(* IEC 61131-3 sources: VFDLib/, 12 files *)

(* ---- VFD.typ ---- *)
(********************************************************************
 * COPYRIGHT -- Automation Resources Group
 ********************************************************************
 * Library: VFDLib
 * File: VFD.typ
 * Author: David Blackburn
 * Created: December 21, 2011
 ********************************************************************
 * Data types of library VFDLib
 ********************************************************************)

TYPE
	VFD_ST_enum :
		(
		VFD_ST_NOTRDYTOSWON := 1,
		VFD_ST_SWONDISABLED,
		VFD_ST_RDYTOSWON,
		VFD_ST_SWON,
		VFD_ST_ENABLED,
		VFD_ST_QUICKSTOPACTIVE,
		VFD_ST_FAULTRXNACTIVE,
		VFD_ST_FAULT,
		VFD_ST_
		);
	VFD_Internal_typ : 	STRUCT
		ScaleIn : Scale_typ;
		ScaleOut : Scale_typ;
		AckResetTimer : TON;
		CMD : VFD_IN_CMD_typ;
	END_STRUCT;
	VFD_TEST_STAT_typ : 	STRUCT
		ActualVelocity : REAL;
		ActualVelocity_RPM : REAL;
		Error : BOOL;
		ErrorID : UINT;
		ErrorString : STRING[VFD_STRLEN_ERROR];
		RdyToSwOn : BOOL;
		SwOn : BOOL;
		OpEnabled : BOOL;
		Fault : BOOL;
		FaultID : UINT;
		VoltageDisabled : BOOL;
		QuickStop : BOOL;
		SwOnDisabled : BOOL;
		AlarmPresent : BOOL;
		RefReached : BOOL;
		State : DINT;
	END_STRUCT;
	VFD_TEST_typ : 	STRUCT
		Enable : BOOL;
		CMD : VFD_IN_CMD_typ;
		PAR : VFD_IN_PAR_typ;
		STAT : VFD_TEST_STAT_typ;
	END_STRUCT;
	VFD_OUT_STAT_Extended_typ : 	STRUCT
		Running : BOOL;
		DCInjection : BOOL;
		Transient : BOOL;
		ThermalOverloadAlarm : BOOL;
		BrakeAlarm : BOOL;
		Accelerating : BOOL;
		Decelerating : BOOL;
		CurrentLimitAlarm : BOOL;
		FastStop : BOOL;
		DirectionReq : BOOL;
	END_STRUCT;
	VFD_OUT_STAT_DriveStatus_typ : 	STRUCT
		RdyToSwOn : BOOL;
		SwOn : BOOL;
		OpEnabled : BOOL;
		Fault : BOOL;
		FaultID : UINT;
		FaultString : STRING[VFD_STRLEN_ERROR];
		VoltageDisabled : BOOL;
		QuickStop : BOOL;
		SwOnDisabled : BOOL;
		AlarmPresent : BOOL;
		RefReached : BOOL;
		RefExceeded : BOOL;
		StopKey : BOOL;
		DirectionOut : BOOL;
	END_STRUCT;
	VFD_OUT_STAT_typ : 	STRUCT
		ActualVelocity : REAL;
		ActualVelocity_RPM : REAL;
		DriveStatus : VFD_OUT_STAT_DriveStatus_typ;
		Extended : VFD_OUT_STAT_Extended_typ;
		State : DINT;
		Error : BOOL;
		ErrorID : UINT;
		ErrorString : STRING[VFD_STRLEN_ERROR];
	END_STRUCT;
	VFD_OUT_typ : 	STRUCT
		STAT : VFD_OUT_STAT_typ;
	END_STRUCT;
	VFD_IN_CFG_Scale_typ : 	STRUCT
		MinUnits : REAL;
		MinRPM : REAL;
		MaxUnits : REAL;
		MaxRPM : REAL;
	END_STRUCT;
	VFD_IN_CFG_typ : 	STRUCT
		Scale : VFD_IN_CFG_Scale_typ; (*2-point motor speed scaling*)
	END_STRUCT;
	VFD_IN_PAR_typ : 	STRUCT
		Velocity : REAL; (*Set motor speed in units.*)
	END_STRUCT;
	VFD_IN_CMD_typ : 	STRUCT
		Power : BOOL; (*Enable motor output*)
		Run : BOOL; (*Run motor at speed*)
		Reverse : BOOL; (*Run in reverse (must also set Run for motion)*)
		AcknowledgeError : BOOL; (*Reset drive faults*)
		Restart : BOOL; (*Restart drive after recovering from a fault*)
	END_STRUCT;
	VFD_IN_typ : 	STRUCT
		CMD : VFD_IN_CMD_typ;
		PAR : VFD_IN_PAR_typ;
		CFG : VFD_IN_CFG_typ;
	END_STRUCT;
	VFD_typ : 	STRUCT
		IN : VFD_IN_typ;
		OUT : VFD_OUT_typ;
		TEST : VFD_TEST_typ;
		IOMap : VFD_IO_typ;
		Encoder : VFD_Encoder_typ;
		Internal : VFD_Internal_typ;
	END_STRUCT;
END_TYPE

(* ---- VFD_IO.typ ---- *)
(*
 * File: VFD_IO.typ
 * Copyright (c) 2023 Loupe
 * https://loupe.team
 *
 * This file is part of VFDLib, licensed under the MIT License.
 *
 *)

TYPE
	VFD_IO_OUT_typ : 	STRUCT
		CMDD_Output : UINT;
		CMI_Output : UINT;
		LFRD_Output : INT;
		IOLR_Output_Bool : ARRAY[0..9] OF BOOL;
		DigitalOutput01 : BOOL;
		EnableCounter : BOOL;
	END_STRUCT;
	VFD_IO_IN_ModuleInfo_typ : 	STRUCT
		SerialNumber : UDINT;
		ModuleID : UINT;
		HardwareVariant : UINT;
		FirmwareVersion : UINT;
		ACPi_ModuleID : UDINT;
		ACPi_SerialNumber : UDINT;
	END_STRUCT;
	VFD_IO_IN_typ : 	STRUCT
		ModuleOK : BOOL;
		ModuleInfo : VFD_IO_IN_ModuleInfo_typ;
		ETAD_Input : UINT;
		ETI_Input : UINT;
		RFRD_Input : INT;
		OTR_Input : INT;
		LCR_Input : UINT;
		THD_Input : UINT;
		THR_Input : UINT;
		IOLR_Input_Bool : ARRAY[0..9] OF BOOL;
		ERRD_Input : UINT;
		LFT_Input : INT;
		StatusDigitalOutput01 : BOOL;
		Counter : DINT;
	END_STRUCT;
	VFD_IO_typ : 	STRUCT
		IN : VFD_IO_IN_typ;
		OUT : VFD_IO_OUT_typ;
	END_STRUCT;
END_TYPE

(* ---- VFDEncoder.typ ---- *)
(*
 * File: VFDEncoder.typ
 * Copyright (c) 2023 Loupe
 * https://loupe.team
 *
 * This file is part of VFDLib, licensed under the MIT License.
 *
 *)

TYPE
	VFD_Encoder_Internal_typ : 	STRUCT
		RTInfo : RTInfo;
		SpeedEst : SpeedEst;
		ScaleOut : Scale_typ;
	END_STRUCT;
	VFD_Encoder_OUT_STAT_typ : 	STRUCT
		Error : BOOL;
	END_STRUCT;
	VFD_Encoder_OUT_typ : 	STRUCT
		SpeedUnits : REAL;
		SpeedCounts : REAL;
		STAT : VFD_Encoder_OUT_STAT_typ;
	END_STRUCT;
	VFD_Encoder_IN_CFG_Scale_typ : 	STRUCT
		MinUnits : REAL;
		MinCounts : REAL;
		MaxUnits : REAL;
		MaxCounts : REAL;
	END_STRUCT;
	VFD_Encoder_IN_CFG_typ : 	STRUCT
		Scale : VFD_Encoder_IN_CFG_Scale_typ;
		tf : REAL;
		deadband : DINT;
		K : REAL;
	END_STRUCT;
	VFD_Encoder_IN_typ : 	STRUCT
		Counter : DINT;
		CFG : VFD_Encoder_IN_CFG_typ;
	END_STRUCT;
	VFD_Encoder_typ : 	STRUCT
		IN : VFD_Encoder_IN_typ;
		OUT : VFD_Encoder_OUT_typ;
		Internal : VFD_Encoder_Internal_typ;
	END_STRUCT;
END_TYPE

(* ---- VFD_EncoderFn_Cyclic.st ---- *)
(********************************************************************
 * COPYRIGHT --  Automation Resources Group
 ********************************************************************
 * Library: VFD_Lib
 * File: VFD_EncoderFn_Cyclic.st
 * Author: David
 * Created: September 09, 2010
 ********************************************************************
 * Implementation of library VFD_Lib
 ********************************************************************)

(********************************************************************)
(* Cyclic function for getting VFD speed from encoder feedback 		*)
(********************************************************************)

(* RTInfo FUB		DONE and TESTED DFB *)
(* SpdEst FUB		DONE and TESTED DFB *)
(* Scaling			DONE and TESTED DFB *)
(* Outputs			DONE and TESTED DFB *)

FUNCTION VFD_EncoderFn_Cyclic

(************************************************************)
(* Set return value to get rid of compile warning 			*)
(************************************************************)

VFD_EncoderFn_Cyclic:=	FALSE;

(************************************************************)
(* Find period using RTInfo FUB					 			*)
(************************************************************)

t.Internal.RTInfo.enable:=	1;

t.Internal.RTInfo();

(************************************************************)
(* SpdEst FUB									 			*)
(************************************************************)

t.Internal.SpeedEst.Position:=	t.IN.Counter;
t.Internal.SpeedEst.T:=			UDINT_TO_REAL(t.Internal.RTInfo.cycle_time) / 1000000.0;	(* sample period [s] *)

(* Default tf to 100ms *)

IF( t.IN.CFG.tf = 0 )THEN
	t.Internal.SpeedEst.tf:=	0.1;
ELSE
	t.Internal.SpeedEst.tf:=	t.IN.CFG.tf;
END_IF

t.Internal.SpeedEst.deadband:=	t.IN.CFG.deadband;
t.Internal.SpeedEst.K:=			t.IN.CFG.K;

t.Internal.SpeedEst();

(************************************************************)
(* Scaling										 			*)
(************************************************************)

t.Internal.ScaleOut.IN.InputValue:=	t.Internal.SpeedEst.Speed_est;

t.Internal.ScaleOut.IN.CFG.Point[0].Input:=		t.IN.CFG.Scale.MinCounts;
t.Internal.ScaleOut.IN.CFG.Point[0].Output:=	t.IN.CFG.Scale.MinUnits;
t.Internal.ScaleOut.IN.CFG.Point[1].Input:=		t.IN.CFG.Scale.MaxCounts;
t.Internal.ScaleOut.IN.CFG.Point[1].Output:=	t.IN.CFG.Scale.MaxUnits;

ScaleFnCyclic( t.Internal.ScaleOut );

(************************************************************)
(* Encoder outputs								 			*)
(************************************************************)

t.OUT.SpeedUnits:=	t.Internal.ScaleOut.OUT.OutputValue;
t.OUT.SpeedCounts:=	t.Internal.SpeedEst.Speed_est;

IF( (t.Internal.RTInfo.status <> 0)			OR
	(t.Internal.ScaleOut.OUT.STAT.Error)	)THEN

	t.OUT.STAT.Error:=	1;

ELSE

	t.OUT.STAT.Error:=	0;

END_IF

END_FUNCTION

(* ---- VFD_GetDriveStatus.st ---- *)
(*
 * File: VFD_GetDriveStatus.st
 * Copyright (c) 2023 Loupe
 * https://loupe.team
 *
 * This file is part of VFDLib, licensed under the MIT License.
 *
 *)

(********************************************************************)
(* This function unpacks the DriveStatus word						*)
(********************************************************************)

(* Functionality			DONE and TESTED DFB 20110512 *)

FUNCTION VFD_GetDriveStatus

(************************************************************)
(* Set return value to get rid of compile warning 			*)
(************************************************************)

VFD_GetDriveStatus:=	FALSE;

(************************************************************)
(* Unpack DriveStatus				 						*)
(************************************************************)

DriveStatus.RdyToSwOn:=			ETAD_Input.0;
DriveStatus.SwOn:=				ETAD_Input.1;
DriveStatus.OpEnabled:=			ETAD_Input.2;
DriveStatus.Fault:=				ETAD_Input.3;
DriveStatus.VoltageDisabled:=	ETAD_Input.4;
DriveStatus.QuickStop:=			ETAD_Input.5;
DriveStatus.SwOnDisabled:=		ETAD_Input.6;
DriveStatus.AlarmPresent:=		ETAD_Input.7;
DriveStatus.RefReached:=		ETAD_Input.10;
DriveStatus.RefExceeded:=		ETAD_Input.11;
DriveStatus.StopKey:=			ETAD_Input.14;
DriveStatus.DirectionOut:=		ETAD_Input.15;

END_FUNCTION

(* ---- VFD_GetExtendedStatus.st ---- *)
(*
 * File: VFD_GetExtendedStatus.st
 * Copyright (c) 2023 Loupe
 * https://loupe.team
 *
 * This file is part of VFDLib, licensed under the MIT License.
 *
 *)

(********************************************************************)
(* This functions unpacks the Extended status word 					*)
(********************************************************************)

(* Functionality		DONE and TESTED DFB 20110512 *)

FUNCTION VFD_GetExtendedStatus

(************************************************************)
(* Set return value to get rid of compile warning 			*)
(************************************************************)

VFD_GetExtendedStatus:=	FALSE;

(************************************************************)
(* Unpack ExtendedStatus				 					*)
(************************************************************)

ExtendedStatus.Running:= 				ETI_Input.4;
ExtendedStatus.DCInjection:= 			ETI_Input.5;
ExtendedStatus.Transient:= 				ETI_Input.6;
ExtendedStatus.ThermalOverloadAlarm:= 	ETI_Input.7;
ExtendedStatus.BrakeAlarm:= 			ETI_Input.8;
ExtendedStatus.Accelerating:= 			ETI_Input.9;
ExtendedStatus.Decelerating:=		 	ETI_Input.10;
ExtendedStatus.CurrentLimitAlarm:= 		ETI_Input.11;
ExtendedStatus.FastStop:= 				ETI_Input.12;
ExtendedStatus.DirectionReq:= 			ETI_Input.15;

END_FUNCTION

(* ---- VFD_SetCMDD_Output_X64.st ---- *)
(********************************************************************
 * COPYRIGHT --  Automation Resources Group
 ********************************************************************
 * Library: VFD_Lib
 * File: VFD_SetCMDD_Output_X64.st
 * Author: blackburnd
 * Created: September 7, 2010
 ********************************************************************
 * Implementation of library VFD_Lib
 ********************************************************************)

(************************************************************************************)
(* This function sets the bits in the control word based on the axis input values.	*)
(************************************************************************************)

(* SwOn, EnableOperation					DONE and TESTED DFB *)
	(* Setting								see VFDFnCyclic.st *)
	(* Resetting							DONE and TESTED DFB *)

(* VoltageDisable							DONE and TESTED DFB *)

(* QuickStop								DONE and TESTED DFB *)

(* FaultReset								DONE and TESTED DFB *)

(* Reverse									DONE and TESTED DFB *)

(* Stop_Stt									DONE and TESTED DFB *)

FUNCTION VFD_SetCMDD_Output_X64

(************************************************************)
(* Set return value to get rid of compile warning 			*)
(************************************************************)

VFD_SetCMDD_Output_X64:=	FALSE;

(****************************************************************************)
(* Switch On and Enable Operation control bits are set in the state machine	*)
(* They are reset here *)

IF( NOT(t.IN.CMD.Power) ) THEN

	t.IOMap.OUT.CMDD_Output:=	BIT_CLR(t.IOMap.OUT.CMDD_Output, VFD_CTRLBIT_SWON);
	t.IOMap.OUT.CMDD_Output:=	BIT_CLR(t.IOMap.OUT.CMDD_Output, VFD_CTRLBIT_ENABLEOPERATION);

END_IF

(****************************************************************************)
(* Set VoltageDisable bit based on enable *)
(* 0 = Disable voltage, 1 = Enable Voltage *)

IF( t.IN.CMD.Power )THEN

	t.IOMap.OUT.CMDD_Output:=	BIT_SET(t.IOMap.OUT.CMDD_Output, VFD_CTRLBIT_DISABLEVOLTAGE);

ELSE

	t.IOMap.OUT.CMDD_Output:=	BIT_CLR(t.IOMap.OUT.CMDD_Output, VFD_CTRLBIT_DISABLEVOLTAGE);

END_IF

(****************************************************************************)
(* Set quickstop control bit (no quickstop functionality supported) *)
(* 0 = Quickstop active, 1 = Quickstop inactive *)

t.IOMap.OUT.CMDD_Output:=	BIT_SET(t.IOMap.OUT.CMDD_Output, VFD_CTRLBIT_QUICKSTOP);

(****************************************************************************)
(* Set Fault Reset and warning reset control bits according to CMD  *)
(* THIS MIGHT ALSO NEED TO BE IN THE STATE MACHINE *)

IF( t.IN.CMD.AcknowledgeError ) THEN

	t.IOMap.OUT.CMDD_Output:=	BIT_SET(t.IOMap.OUT.CMDD_Output, VFD_CTRLBIT_FAULTRESET);

ELSE

	t.IOMap.OUT.CMDD_Output:=	BIT_CLR(t.IOMap.OUT.CMDD_Output, VFD_CTRLBIT_FAULTRESET);

END_IF

(****************************************************************************)
(* Set reverse bit based on command *)
(* THIS MIGHT ALSO NEED TO BE IN THE STATE MACHINE *)

IF( t.IN.CMD.Reverse ) THEN

	t.IOMap.OUT.CMDD_Output:=	BIT_SET(t.IOMap.OUT.CMDD_Output, VFD_CTRLBIT_REV);

ELSE

	t.IOMap.OUT.CMDD_Output:=	BIT_CLR(t.IOMap.OUT.CMDD_Output, VFD_CTRLBIT_REV);

END_IF

(****************************************************************************)
(* Set Stop bit based on command *)
(* THIS MIGHT ALSO NEED TO BE IN THE STATE MACHINE *)

IF( t.IN.CMD.Run ) THEN

	t.IOMap.OUT.CMDD_Output:=	BIT_CLR(t.IOMap.OUT.CMDD_Output, VFD_CTRLBIT_STOP_STT);

ELSE

	t.IOMap.OUT.CMDD_Output:=	BIT_SET(t.IOMap.OUT.CMDD_Output, VFD_CTRLBIT_STOP_STT);

END_IF

END_FUNCTION

(* ---- VFD_SetFaultString.st ---- *)
(********************************************************************
 * COPYRIGHT --  Automation Resources Group
 ********************************************************************
 * Library: VFD_Lib
 * File: VFD_SetFaultString.st
 * Author: David
 * Created: October 12, 2010
 ********************************************************************
 * Implementation of library VFD_Lib
 ********************************************************************)

(************************************************************************)
(* This function sets the error text based on the LFT fault ID input.	*)
(************************************************************************)

(* Functionality		DONE and TESTED DFB *)

FUNCTION VFD_SetFaultString

(************************************************************)
(* Set return value to get rid of compile warning 			*)
(************************************************************)

VFD_SetFaultString:=	FALSE;

(* Set FaultString *)

CASE ID OF

	0:	String:=	'"nOF": No fault code saved';
	3:	String:=	'"CFF": Incorrect configuration (parameters)';
	4:	String:=	'"CFI": Invalid configuration (parameters)';
	5:	String:=	'"SLF": Modbus communication interruption';
	6:	String:=	'"ILF": Internal communication interruption';
	7:	String:=	'"CnF": Communication option card';
	8:	String:=	'"EPF": External fault';
	9:	String:=	'"OCF": Overcurrent';
	10:	String:=	'"CrF": Capacitor pre-charge';
	13:	String:=	'"LFF": 4 - 20 mA loss';
	16:	String:=	'"OHF": Drive overheating';
	17:	String:=	'"OLF": Motor overload';
	18:	String:=	'"ObF": DC bus overvoltage';
	19:	String:=	'"OSF": Line supply overvoltage';
	20:	String:=	'"OPF": Motor phase loss';
	21:	String:=	'"PHF": Line phase loss';
	22:	String:=	'"USF": Line supply undervoltage';
	23:	String:=	'"OCF": Motor short-circuit (phase to phase)';
	24:	String:=	'"SOF": Motor overspeed';
	25:	String:=	'"tnF": Auto-tuning was unsuccessful';
	26:	String:=	'"IF1": Unknown rating';
	27:	String:=	'"IF2": MMI card';
	28:	String:=	'"IF3": MMI communication';
	29:	String:=	'"IF4": Industrial EEPROM';
	30:	String:=	'"EEF": EEPROM memory';
	31:	String:=	'"OCF": Impeding short-circuit';
	32:	String:=	'"SCF": Motor short-circuit (to ground)';
	33:	String:=	'"OPF": Motor phase loss - 3 phases';
	34:	String:=	'"COF": Communication interruption, fault line 2 (CANopen)';
	35:	String:=	'"bLF": Brake control';
	36:	String:=	'"OCF": Power module, specific to 15kW drives';
	55:	String:=	'"SCF": Power module or motor short-circuit, detected at power up.';
	ELSE String:=	'Invalid FaultID';

END_CASE

END_FUNCTION

(* ---- VFD_SetState.st ---- *)
(*
 * File: VFD_SetState.st
 * Copyright (c) 2023 Loupe
 * https://loupe.team
 *
 * This file is part of VFDLib, licensed under the MIT License.
 *
 *)

(********************************************************************)
(* This function sets the state based on the status bits.			*)
(********************************************************************)

(* VFD_ST_NOTRDYTOSWON				DONE and TESTED DFB 20110512 *)
(* VFD_ST_SWONDISABLED				DONE and TESTED DFB 20110512 *)
(* VFD_ST_RDYTOSWON					DONE and TESTED DFB 20110512 *)
(* VFD_ST_SWON						DONE and TESTED DFB 20110512 *)
(* VFD_ST_ENABLED					DONE and TESTED DFB 20110512 *)
(* VFD_ST_QUICKSTOPACTIVE			DONE and TESTED DFB 20110512 *)
(* VFD_ST_FAULTRXNACTIVE			DONE and TESTED DFB 20110512 *)
(* VFD_ST_FAULT						DONE and TESTED DFB 20110512 *)

FUNCTION VFD_SetState

(************************************************************)
(* Set return value to get rid of compile warning 			*)
(************************************************************)

VFD_SetState:=	FALSE;

(************************************************************)
(* Set state 												*)
(************************************************************)

IF( 	(t.DriveStatus.RdyToSwOn = 0)
	AND	(t.DriveStatus.SwOn = 0)
	AND	(t.DriveStatus.OpEnabled = 0)
	AND	(t.DriveStatus.Fault = 0)
	AND	(t.DriveStatus.SwOnDisabled = 0)
	)THEN

	t.State:=	VFD_ST_NOTRDYTOSWON;

ELSIF(		(t.DriveStatus.RdyToSwOn = 0)
		AND	(t.DriveStatus.SwOn = 0)
		AND	(t.DriveStatus.OpEnabled = 0)
		AND	(t.DriveStatus.Fault = 0)
		AND	(t.DriveStatus.SwOnDisabled = 1)
		)THEN

	t.State:=	VFD_ST_SWONDISABLED;

ELSIF(		(t.DriveStatus.RdyToSwOn = 1)
		AND	(t.DriveStatus.SwOn = 0)
		AND	(t.DriveStatus.OpEnabled = 0)
		AND	(t.DriveStatus.Fault = 0)
		AND	(t.DriveStatus.QuickStop = 1)
		AND	(t.DriveStatus.SwOnDisabled = 0)
		)THEN

	t.State:=	VFD_ST_RDYTOSWON;

ELSIF(		(t.DriveStatus.RdyToSwOn = 1)
		AND	(t.DriveStatus.SwOn = 1)
		AND	(t.DriveStatus.OpEnabled = 0)
		AND	(t.DriveStatus.Fault = 0)
		AND	(t.DriveStatus.QuickStop = 1)
		AND	(t.DriveStatus.SwOnDisabled = 0)
		)THEN

	t.State:=	VFD_ST_SWON;

ELSIF(		(t.DriveStatus.RdyToSwOn = 1)
		AND	(t.DriveStatus.SwOn = 1)
		AND	(t.DriveStatus.OpEnabled = 1)
		AND	(t.DriveStatus.Fault = 0)
		AND	(t.DriveStatus.QuickStop = 1)
		AND	(t.DriveStatus.SwOnDisabled = 0)
		)THEN

	t.State:=	VFD_ST_ENABLED;

ELSIF(	(t.DriveStatus.RdyToSwOn = 1)
		AND	(t.DriveStatus.SwOn = 1)
		AND	(t.DriveStatus.OpEnabled = 1)
		AND	(t.DriveStatus.Fault = 0)
		AND	(t.DriveStatus.QuickStop = 0)
		AND	(t.DriveStatus.SwOnDisabled = 0)
		)THEN

	t.State:=	VFD_ST_QUICKSTOPACTIVE;

ELSIF(		(t.DriveStatus.RdyToSwOn = 1)
		AND	(t.DriveStatus.SwOn = 1)
  		AND	(t.DriveStatus.OpEnabled = 1)
		AND	(t.DriveStatus.Fault = 1)
		AND	(t.DriveStatus.SwOnDisabled = 0)
		)THEN

	t.State:=	VFD_ST_FAULTRXNACTIVE;

ELSIF(	(t.DriveStatus.RdyToSwOn = 0)
		AND	(t.DriveStatus.SwOn = 0)
		AND	(t.DriveStatus.OpEnabled = 0)
		AND	(t.DriveStatus.Fault = 1)
		AND	(t.DriveStatus.SwOnDisabled = 0)
		)THEN

	t.State:=	VFD_ST_FAULT;

END_IF

END_FUNCTION

(* ---- VFDFn_Cyclic.st ---- *)
(********************************************************************
 * COPYRIGHT --  Automation Resources Group
 ********************************************************************
 * Library: VFD_Lib
 * File: VFDFn_Cyclic.st
 * Author: David
 * Created: September 07, 2010
 ********************************************************************
 * Implementation of library VFD_Lib
 ********************************************************************)

(********************************************************************)
(* Cyclic function for controlling one VFD 							*)
(********************************************************************)

(* Handling TEST interface						DONE and TESTED DFB 20110512 *)
	(* CMD, PAR									DONE and TESTED DFB 20110511 *)
	(* STAT										DONE and TESTED DFB 20110512 *)

(* Getting status								see VFD_GetStatusFromStatusUINT.st *)

(* Setting machine state						see VFD_SetState.st *)

(* Setting Control Bits							see VFD_SetControlUINT_XXX.st *)
	(* SwOn, Enable	Setting						DONE and TESTED DFB *)

(* Operation when enabled						DONE and TESTED DFB *)

(* Speed scaling								DONE and TESTED DFB *)
	(* Input									DONE and TESTED DFB *)
	(* Output									DONE and TESTED DFB *)
	(* Error checking							DONE and TESTED DFB *)

(* Populating FaultID							DONE and TESTED DFB 20110512 *)
(* Populating FaultString						see VFD_SetFaultString.st *)

(* Encoder handling								see VFD_EncoderFnCyclic.st *)

(* Error reporting								DONE and TESTED DFB 20111220 *)

(* Error acknowledgement						DONE not tested *)
	(* Drive faults								DONE not tested *)
	(* Scaling errors							DONE and TESTED DFB 20111220 *)

FUNCTION VFDFn_Cyclic

(************************************************************)
(* Set return value to get rid of compile warning 			*)
(************************************************************)

VFDFn_Cyclic:=	FALSE;

(****************************************************)
(* Handle TEST interface							*)
(****************************************************)

IF( t.TEST.Enable )THEN

	(* Overwrite IN.CMDs and IN.PARs while in TEST mode *)

	t.IN.CMD:=	t.TEST.CMD;
	t.IN.PAR:=	t.TEST.PAR;

ELSE

    (* Clear TEST.CMDs and load TEST.PARs from machine while not in TEST mode *)

	brsmemset( ADR(t.TEST.CMD), 0, SIZEOF(t.TEST.CMD));
	t.TEST.PAR:=	t.IN.PAR;

END_IF

(************************************************************)
(* Handle internal CMD image resets							*)
(************************************************************)

IF( NOT(t.IN.CMD.Restart) )THEN

	t.Internal.CMD.Restart:=	0;

END_IF

(************************************************************)
(* Set control bits accordingly								*)
(************************************************************)

VFD_SetCMDD_Output_X64( t );

(************************************************************)
(* Get DriveStatus and Extended status						*)
(************************************************************)

VFD_GetDriveStatus( t.IOMap.IN.ETAD_Input, t.OUT.STAT.DriveStatus );
VFD_GetExtendedStatus( t.IOMap.IN.ETI_Input, t.OUT.STAT.Extended );

(************************************************************)
(* Main State Machine										*)
(************************************************************)

(* Set State based on status bits *)

VFD_SetState( t.OUT.STAT );

CASE t.OUT.STAT.State OF

	VFD_ST_NOTRDYTOSWON:

	VFD_ST_SWONDISABLED:

		(* It is possible to get to this state through a fault condition without disabling the VFD. *)
		(* If this is the case, then bits VFD_CTRLBIT_SWON and VFD_CTRLBIT_ENABLEOPERATION will not be reset. *)
		(* This will make it impossible to leave this state. *)
		(* So, handle a Reset CMD in this state to reset those two bits to get back to VFD_ST_ENABLED. *)

		IF( t.IN.CMD.Restart AND NOT(t.Internal.CMD.Restart) )THEN

  			t.Internal.CMD.Restart:=	1;

			t.IOMap.OUT.CMDD_Output:=	BIT_CLR(t.IOMap.OUT.CMDD_Output, VFD_CTRLBIT_SWON);
			t.IOMap.OUT.CMDD_Output:=	BIT_CLR(t.IOMap.OUT.CMDD_Output, VFD_CTRLBIT_ENABLEOPERATION);

		END_IF

	VFD_ST_RDYTOSWON:

		(* If enabled, set SwOn bit *)

		IF( t.IN.CMD.Power ) THEN

			t.IOMap.OUT.CMDD_Output:=	BIT_SET(t.IOMap.OUT.CMDD_Output, VFD_CTRLBIT_SWON);

		END_IF

	VFD_ST_SWON:

		(* If enabled, set EnableOp bit *)

		IF( t.IN.CMD.Power ) THEN

			t.IOMap.OUT.CMDD_Output:=		BIT_SET(t.IOMap.OUT.CMDD_Output, VFD_CTRLBIT_ENABLEOPERATION);

		END_IF

	VFD_ST_ENABLED:

	VFD_ST_QUICKSTOPACTIVE:

	VFD_ST_FAULTRXNACTIVE:

	VFD_ST_FAULT:

END_CASE

(************************************************************)
(* Actual speed input scaling (RPM to Units)				*)
(************************************************************)

t.Internal.ScaleIn.IN.InputValue:=	INT_TO_REAL( t.IOMap.IN.RFRD_Input );

t.Internal.ScaleIn.IN.CFG.Point[0].Input	:=	t.IN.CFG.Scale.MinRPM;
t.Internal.ScaleIn.IN.CFG.Point[0].Output	:=	t.IN.CFG.Scale.MinUnits;
t.Internal.ScaleIn.IN.CFG.Point[1].Input	:=	t.IN.CFG.Scale.MaxRPM;
t.Internal.ScaleIn.IN.CFG.Point[1].Output	:=	t.IN.CFG.Scale.MaxUnits;

ScaleFnCyclic( t.Internal.ScaleIn );

t.OUT.STAT.ActualVelocity:=		t.Internal.ScaleIn.OUT.OutputValue;
t.OUT.STAT.ActualVelocity_RPM:=	INT_TO_REAL( t.IOMap.IN.RFRD_Input );

(************************************************************)
(* Set speed output scaling (Units to RPM)					*)
(************************************************************)

t.Internal.ScaleOut.IN.InputValue:=	t.IN.PAR.Velocity;

t.Internal.ScaleOut.IN.CFG.Point[0].Input	:=	t.IN.CFG.Scale.MinUnits;
t.Internal.ScaleOut.IN.CFG.Point[0].Output	:=	t.IN.CFG.Scale.MinRPM;
t.Internal.ScaleOut.IN.CFG.Point[1].Input	:=	t.IN.CFG.Scale.MaxUnits;
t.Internal.ScaleOut.IN.CFG.Point[1].Output	:=	t.IN.CFG.Scale.MaxRPM;

ScaleFnCyclic( t.Internal.ScaleOut );

t.IOMap.OUT.LFRD_Output:=	REAL_TO_INT( t.Internal.ScaleOut.OUT.OutputValue );

(************************************************************)
(* Set FaultID and FaultString								*)
(************************************************************)

t.OUT.STAT.DriveStatus.FaultID:=	t.IOMap.IN.LFT_Input;

VFD_SetFaultString( t.OUT.STAT.DriveStatus.FaultID, t.OUT.STAT.DriveStatus.FaultString );

(************************************************************)
(* Encoder handling											*)
(************************************************************)

t.IOMap.OUT.EnableCounter:=	1;

t.Encoder.IN.Counter:=		t.IOMap.IN.Counter;

VFD_EncoderFn_Cyclic( t.Encoder );

(************************************************************)
(* Error reporting and acknowledgement						*)
(************************************************************)

(* Handle CMD.AcknowledgeError - doing this before
	setting Error status gets rid of the one scan toggle on Error. *)

(* Wait 50ms before resetting CMD.AcknowledgeError and clearing
	error status. This will allow the VFD time to respond appropriately *)

t.Internal.AckResetTimer.IN:=	t.IN.CMD.AcknowledgeError;
t.Internal.AckResetTimer.PT:=	T#50ms;

t.Internal.AckResetTimer();

IF( t.Internal.AckResetTimer.Q )THEN

	t.IN.CMD.AcknowledgeError:=	0;

	t.OUT.STAT.Error:=			0;
	t.OUT.STAT.ErrorID:=		0;
	t.OUT.STAT.ErrorString:=	'';

END_IF

(* Set Error status *)

IF( t.OUT.STAT.DriveStatus.Fault )THEN

	t.OUT.STAT.Error:=			1;
	t.OUT.STAT.ErrorID:=		t.OUT.STAT.DriveStatus.FaultID;
	t.OUT.STAT.ErrorString:=	t.OUT.STAT.DriveStatus.FaultString;

ELSIF( 		t.Internal.ScaleIn.OUT.STAT.Error
		OR	t.Internal.ScaleOut.OUT.STAT.Error
		)THEN

	t.OUT.STAT.Error:=			1;
	t.OUT.STAT.ErrorString:=	'Speed scaling error. Check IN.CFG.Scale.';

ELSIF( t.Encoder.OUT.STAT.Error )THEN

	t.OUT.STAT.Error:=			1;
	t.OUT.STAT.ErrorString:=	'Encoder scaling error. Check Encoder.IN.CFG.Scale.';

END_IF

(********************************************************************)
(* Map TEST.STAT items												*)
(********************************************************************)

t.TEST.STAT.ActualVelocity:=		t.OUT.STAT.ActualVelocity;
t.TEST.STAT.ActualVelocity_RPM:=	t.OUT.STAT.ActualVelocity_RPM;
t.TEST.STAT.Error:=					t.OUT.STAT.Error;
t.TEST.STAT.ErrorID:=				t.OUT.STAT.ErrorID;
t.TEST.STAT.ErrorString:=			t.OUT.STAT.ErrorString;
t.TEST.STAT.RdyToSwOn:=				t.OUT.STAT.DriveStatus.RdyToSwOn;
t.TEST.STAT.SwOn:=					t.OUT.STAT.DriveStatus.SwOn;
t.TEST.STAT.OpEnabled:=				t.OUT.STAT.DriveStatus.OpEnabled;
t.TEST.STAT.Fault:=					t.OUT.STAT.DriveStatus.Fault;
t.TEST.STAT.FaultID:=				t.OUT.STAT.DriveStatus.FaultID;
t.TEST.STAT.VoltageDisabled:=		t.OUT.STAT.DriveStatus.VoltageDisabled;
t.TEST.STAT.QuickStop:=				t.OUT.STAT.DriveStatus.QuickStop;
t.TEST.STAT.SwOnDisabled:=			t.OUT.STAT.DriveStatus.SwOnDisabled;
t.TEST.STAT.AlarmPresent:=			t.OUT.STAT.DriveStatus.AlarmPresent;
t.TEST.STAT.RefReached:=			t.OUT.STAT.DriveStatus.RefReached;
t.TEST.STAT.State:=					t.OUT.STAT.State;

END_FUNCTION

(* ---- VFDLib.fun ---- *)
(*
 * File: VFDLib.fun
 * Copyright (c) 2023 Loupe
 * https://loupe.team
 *
 * This file is part of VFDLib, licensed under the MIT License.
 *
 *)

FUNCTION VFDFn_Cyclic : BOOL (*Cyclic function for controlling one VFD*)
	VAR_IN_OUT
		t : VFD_typ; (*VFD control object*)
	END_VAR
END_FUNCTION

FUNCTION VFD_SetCMDD_Output_X64 : BOOL (*This function sets the bits in the control word based on the axis input values*)
	VAR_IN_OUT
		t : VFD_typ; (*VFD control object*)
	END_VAR
END_FUNCTION

FUNCTION VFD_GetDriveStatus : BOOL (*This function unpacks the DriveStatus word*)
	VAR_INPUT
		ETAD_Input : UINT; (*DriveStatus word*)
	END_VAR
	VAR_IN_OUT
		DriveStatus : VFD_OUT_STAT_DriveStatus_typ; (*DriveStatus structure*)
	END_VAR
END_FUNCTION

FUNCTION VFD_GetExtendedStatus : BOOL (*This functions unpacks the Extended status word*)
	VAR_INPUT
		ETI_Input : UINT; (*Drive Extended status word*)
	END_VAR
	VAR_IN_OUT
		ExtendedStatus : VFD_OUT_STAT_Extended_typ; (*Extended status structure*)
	END_VAR
END_FUNCTION

FUNCTION VFD_SetState : BOOL (*This function sets the state based on the status bits*)
	VAR_IN_OUT
		t : VFD_OUT_STAT_typ; (*VFD status output structure*)
	END_VAR
END_FUNCTION

FUNCTION VFD_SetFaultString : BOOL (*This function sets the error text based on the LFT fault ID input.*)
	VAR_INPUT
		ID : UINT; (*FaultID*)
	END_VAR
	VAR_IN_OUT
		String : STRING[80]; (*FaultString*)
	END_VAR
END_FUNCTION

FUNCTION VFD_EncoderFn_Cyclic : BOOL (*Cyclic function for getting VFD speed from encoder feedback*)
	VAR_IN_OUT
		t : VFD_Encoder_typ; (*VFD_Encoder control object*)
	END_VAR
END_FUNCTION

(* ---- VFDLib.var ---- *)
(********************************************************************
 * COPYRIGHT --  Automation Resources Group
 ********************************************************************
 * Library: VFD_Lib
 * File: VFD_Lib.var
 * Author: David
 * Created: September 03, 2010
 ********************************************************************
 * Constants of library VFD_Lib
 ********************************************************************)
(*Control Word Bits*)
VAR CONSTANT
	VFD_STRLEN_ERROR : USINT := 80;
	VFD_CTRLBIT_SWON : USINT := 0;
	VFD_CTRLBIT_DISABLEVOLTAGE : USINT := 1;
	VFD_CTRLBIT_QUICKSTOP : USINT := 2;
	VFD_CTRLBIT_ENABLEOPERATION : USINT := 3;
	VFD_CTRLBIT_FAULTRESET : USINT := 7;
	VFD_CTRLBIT_REV : USINT := 11;
	VFD_CTRLBIT_STOP_STT : USINT := 12;
END_VAR
